Staubli VAL3: iLevel4.pgx

public program iLevel4(num& nNum[] (dimensions=1))
begin
  nNum=dioGet(iLevel4)
end
